FUNCTION_BLOCK L3_SetupRouterF (* Basic Function Block Type *)
  (* Standard: 61499-2 *)
  (* Version 0.0, 2014-11-19, 4DIAC-IDE, 4DIAC-Consortium *)
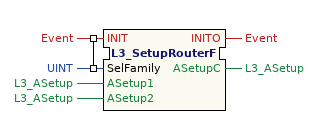
  EVENT_INPUT
    INIT WITH SelFamily; (* Initialization Request *)
  END_EVENT
  EVENT_OUTPUT
    INITO; (* Initialization Confirm *)
  END_EVENT
  VAR_INPUT
    SelFamily : UINT; (* Routing condition *)
  END_VAR
  SOCKETS
    ASetup1 : L3_ASetup;
    ASetup2 : L3_ASetup;
  END_SOCKETS
  PLUGS
    ASetupC : L3_ASetup;
  END_PLUGS
  VAR
    i : USINT; (* loop variable *)
    Select : BOOL; (* Routing cariable *)
  END_VAR
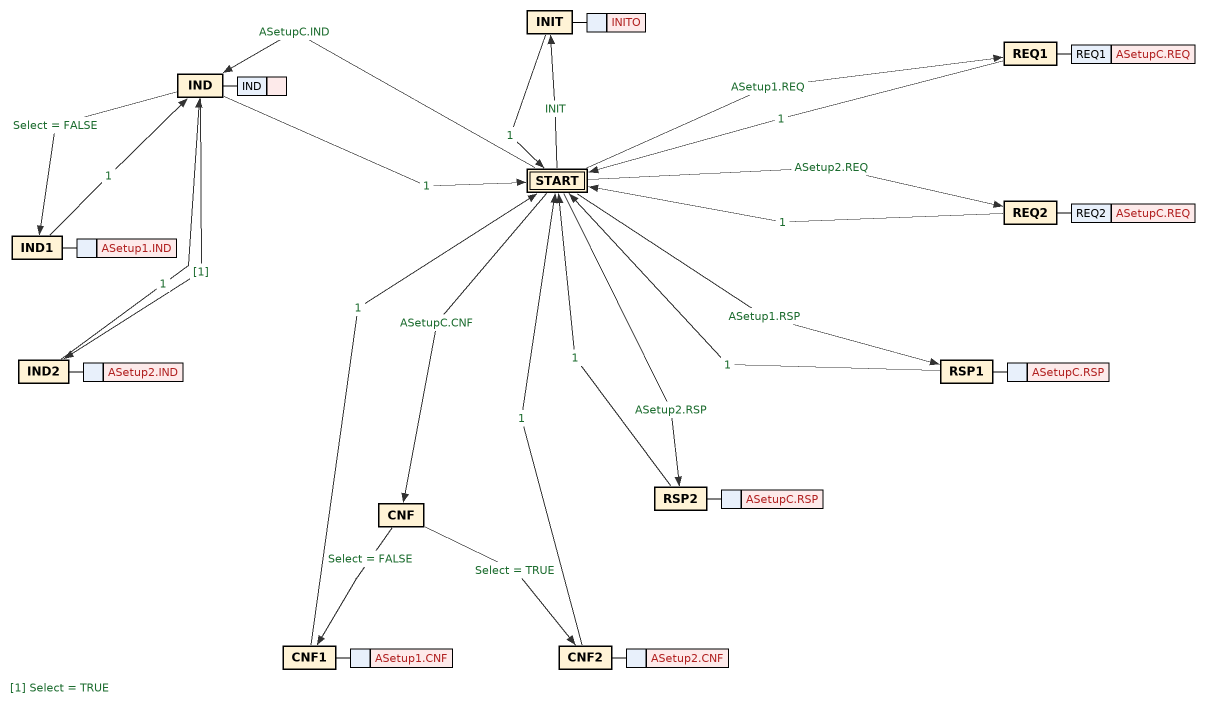
  EC_STATES
    START; (* Initial State *)
    INIT : -> INITO; (* Initialization *)
    REQ1 : REQ1 -> ASetupC.REQ; (* Normal execution *)
    REQ2 : REQ2 -> ASetupC.REQ;
    RSP1 : -> ASetupC.RSP;
    RSP2 : -> ASetupC.RSP;
    CNF;
    CNF1 : -> ASetup1.CNF;
    CNF2 : -> ASetup2.CNF;
    IND : IND;
    IND1 : -> ASetup1.IND;
    IND2 : -> ASetup2.IND;
  END_STATES
  EC_TRANSITIONS
    START TO INIT := INIT;
    INIT TO START := 1;
    START TO REQ1 := ASetup1.REQ;
    REQ1 TO START := 1;
    START TO REQ2 := ASetup2.REQ;
    REQ2 TO START := 1;
    START TO RSP1 := ASetup1.RSP;
    RSP1 TO START := 1;
    START TO RSP2 := ASetup2.RSP;
    RSP2 TO START := 1;
    START TO CNF := ASetupC.CNF;
    CNF TO CNF1 := Select = FALSE;
    CNF TO CNF2 := Select = TRUE;
    CNF1 TO START := 1;
    CNF2 TO START := 1;
    START TO IND := ASetupC.IND;
    IND TO START := 1;
    IND TO IND1 := Select = FALSE;
    IND1 TO IND := 1;
    IND TO IND2 := Select = TRUE;
    IND2 TO IND := 1;
  END_TRANSITIONS
  ALGORITHM REQ1 IN ST: (* Normally executed algorithm *)
FOR i:=0 TO 2 DO
	ASetupC.PartInfoP[i] :=ASetup1.PartInfoP[i];
END_FOR;
ASetupC.MID := ASetup1.MID;
FOR i:=0 TO 19 DO
	ASetupC.OPIDS[i] := ASetup1.OPIDS[i];
	ASetupC.OPParams[i] := ASetup1.OPParams[i];
END_FOR;
ASetupC.Fixture := ASetup1.Fixture;
  END_ALGORITHM
  ALGORITHM REQ2 IN ST: (* new algorithm *)
FOR i:=0 TO 2 DO
	ASetupC.PartInfoP[i] :=ASetup2.PartInfoP[i];
END_FOR;
ASetupC.MID := ASetup2.MID;
FOR i:=0 TO 19 DO
	ASetupC.OPIDS[i] := ASetup2.OPIDS[i];
	ASetupC.OPParams[i] := ASetup2.OPParams[i];
END_FOR;
ASetupC.Fixture := ASetup2.Fixture;
  END_ALGORITHM
  ALGORITHM RSP1 IN ST: (* new algorithm *)
ASetupC.MID := ASetup1.MID;
  END_ALGORITHM
  ALGORITHM RSP2 IN ST: (* new algorithm *)
ASetupC.MID := ASetup2.MID;
  END_ALGORITHM
  ALGORITHM CNF IN ST: (* new algorithm *)
IF ASetupC.PartInfoS[1] = SelFamily THEN
	Select := TRUE;
	ASetup2.PartInfoS[0] := ASetupC.PartInfoS[0];
	ASetup2.PartInfoS[1] := ASetupC.PartInfoS[1];
	ASetup2.PartInfoS[2] := ASetupC.PartInfoS[2];
ELSE
	Select := FALSE;
	ASetup1.PartInfoS[0] := ASetupC.PartInfoS[0];
	ASetup1.PartInfoS[1] := ASetupC.PartInfoS[1];
	ASetup1.PartInfoS[2] := ASetupC.PartInfoS[2];
END_IF;
  END_ALGORITHM
  ALGORITHM IND IN ST: (* new algorithm *)
IF ASetupC.PartInfoS[1] = SelFamily THEN
	Select := TRUE;
	ASetup2.PartInfoS[0] := ASetupC.PartInfoS[0];
	ASetup2.PartInfoS[1] := ASetupC.PartInfoS[1];
	ASetup2.PartInfoS[2] := ASetupC.PartInfoS[2];
	ASetup2.ENDID := ASetupC.ENDID;
ELSE
	Select := FALSE;
	ASetup1.PartInfoS[0] := ASetupC.PartInfoS[0];
	ASetup1.PartInfoS[1] := ASetupC.PartInfoS[1];
	ASetup1.PartInfoS[2] := ASetupC.PartInfoS[2];
	ASetup1.ENDID := ASetupC.ENDID;
END_IF;
  END_ALGORITHM
END_FUNCTION_BLOCK
